// TIA Portal V15.1 export
// export: Created 2024-05-17T05:38:58.0411928Z, ExportSetting WithDefaults, DisplayName Totally Integrated Automation Portal, DisplayVersion V15.1 Update 5, DisplayName TIA Portal Openness, DisplayVersion V15.1 Update 5, DisplayName SINAMICS Startdrive Advanced, DisplayVersion V15.1, DisplayName G130, G150, S120, S150, SINAMICS MV, S210, DisplayVersion V15.1, DisplayName G110M, G120, G120C, G120D, G120P, DisplayVersion V15.1, DisplayName STEP 7 Professional, DisplayVersion V15.1 Update 5, DisplayName STEP 7 Safety, DisplayVersion V15.1, DisplayName WinCC Professional, DisplayVersion V15.1 Update 5, DisplayName SIMATIC Visualization Architect, DisplayVersion V15.1
FUNCTION "209210ZMS012Modes" : Void   // FC311, FBD
TITLE = 209210ZMS012 Modes
{ S7_Optimized_Access := 'FALSE' }
AUTHOR : VCC
FAMILY : Local
NAME : Local
VERSION : 0.1
// stored: AutoNumber false, IsIECCheckEnabled false, SetENOAutomatically False, UDAEnableTagReadback false
   VAR_OUTPUT
      O_AlarmA : Bool;   // Alarm A
      O_AlarmB : Bool;   // Alarm B
      O_AlarmC : Bool;   // Alarm C
      O_AlarmD : Bool;   // Alarm D
      O_AlarmABCondition : Bool;   // Alarms resetable
      H_IAnim : Word;   // Animation bits to Icon in WinCC
   END_VAR
   VAR_TEMP
      NotUsed : Bool;
   END_VAR
BEGIN

REGION Network 1: **** 1 - Inputs **** General Functions
   // General Functions
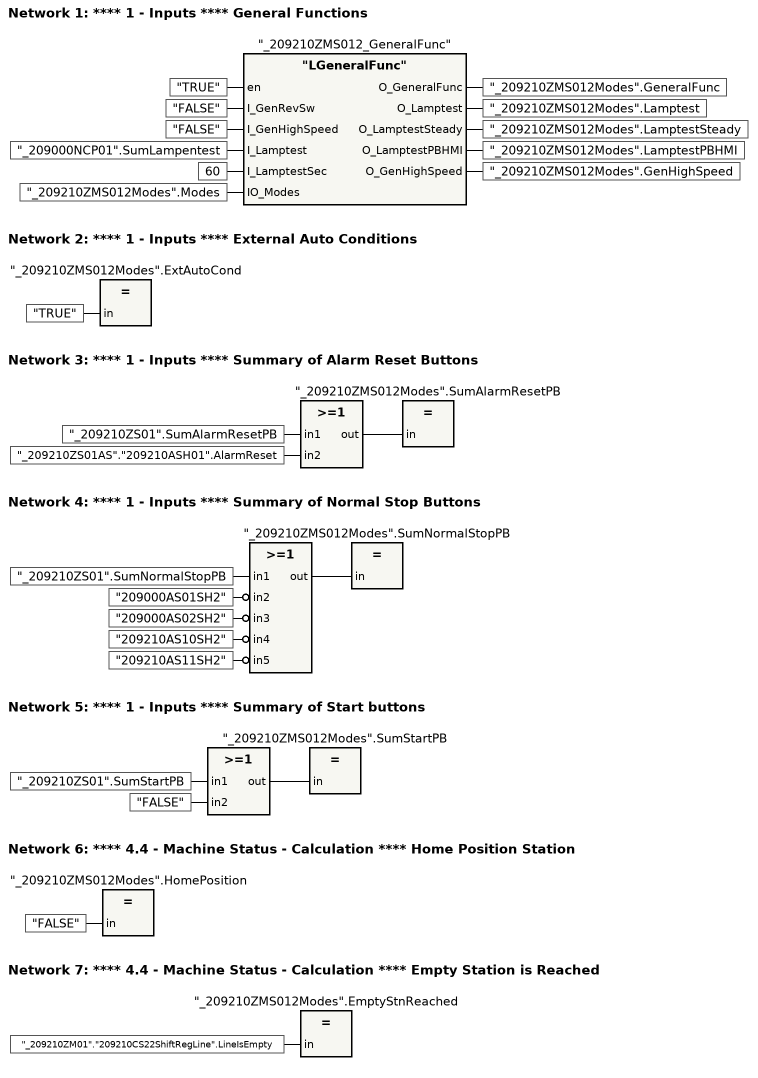
   IF "TRUE" THEN
       "_209210ZMS012_GeneralFunc"(I_GenRevSw := "FALSE",   // "LGeneralFunc"
                               I_GenHighSpeed := "FALSE",
                               I_Lamptest := "_209000NCP01".SumLampentest,
                               I_LamptestSec := 60,
                               IO_Modes := "_209210ZMS012Modes".Modes,
                               O_GeneralFunc => "_209210ZMS012Modes".GeneralFunc,
                               O_Lamptest => "_209210ZMS012Modes".Lamptest,
                               O_LamptestSteady => "_209210ZMS012Modes".LamptestSteady,
                               O_LamptestPBHMI => "_209210ZMS012Modes".LamptestPBHMI,
                               O_GenHighSpeed => "_209210ZMS012Modes".GenHighSpeed);
   END_IF;
END_REGION

REGION Network 2: **** 1 - Inputs **** External Auto Conditions
   "_209210ZMS012Modes".ExtAutoCond := "TRUE";
END_REGION

REGION Network 3: **** 1 - Inputs **** Summary of Alarm Reset Buttons
   // Summary of Alarm Reset Buttons
   "_209210ZMS012Modes".SumAlarmResetPB := "_209210ZS01".SumAlarmResetPB OR "_209210ZS01AS"."209210ASH01".AlarmReset;
END_REGION

REGION Network 4: **** 1 - Inputs **** Summary of Normal Stop Buttons
   // Summary of Normal Stop Buttons
   "_209210ZMS012Modes".SumNormalStopPB := "_209210ZS01".SumNormalStopPB OR NOT "209000AS01SH2" OR NOT "209000AS02SH2" OR NOT "209210AS10SH2" OR NOT "209210AS11SH2";
END_REGION

REGION Network 5: **** 1 - Inputs **** Summary of Start buttons
   // Summary of Start buttons
   "_209210ZMS012Modes".SumStartPB := "_209210ZS01".SumStartPB OR "FALSE";
END_REGION

REGION Network 6: **** 4.4 - Machine Status - Calculation **** Home Position Station
   // Home position
   "_209210ZMS012Modes".HomePosition := "FALSE";
END_REGION

REGION Network 7: **** 4.4 - Machine Status - Calculation **** Empty Station is Reached
   // Empty Station
   "_209210ZMS012Modes".EmptyStnReached := "_209210ZM01"."209210CS22ShiftRegLine".LineIsEmpty;
END_REGION

REGION Network 8: **** 4.5 - Machine Status - Modes **** Mode selector
   // Mode selector
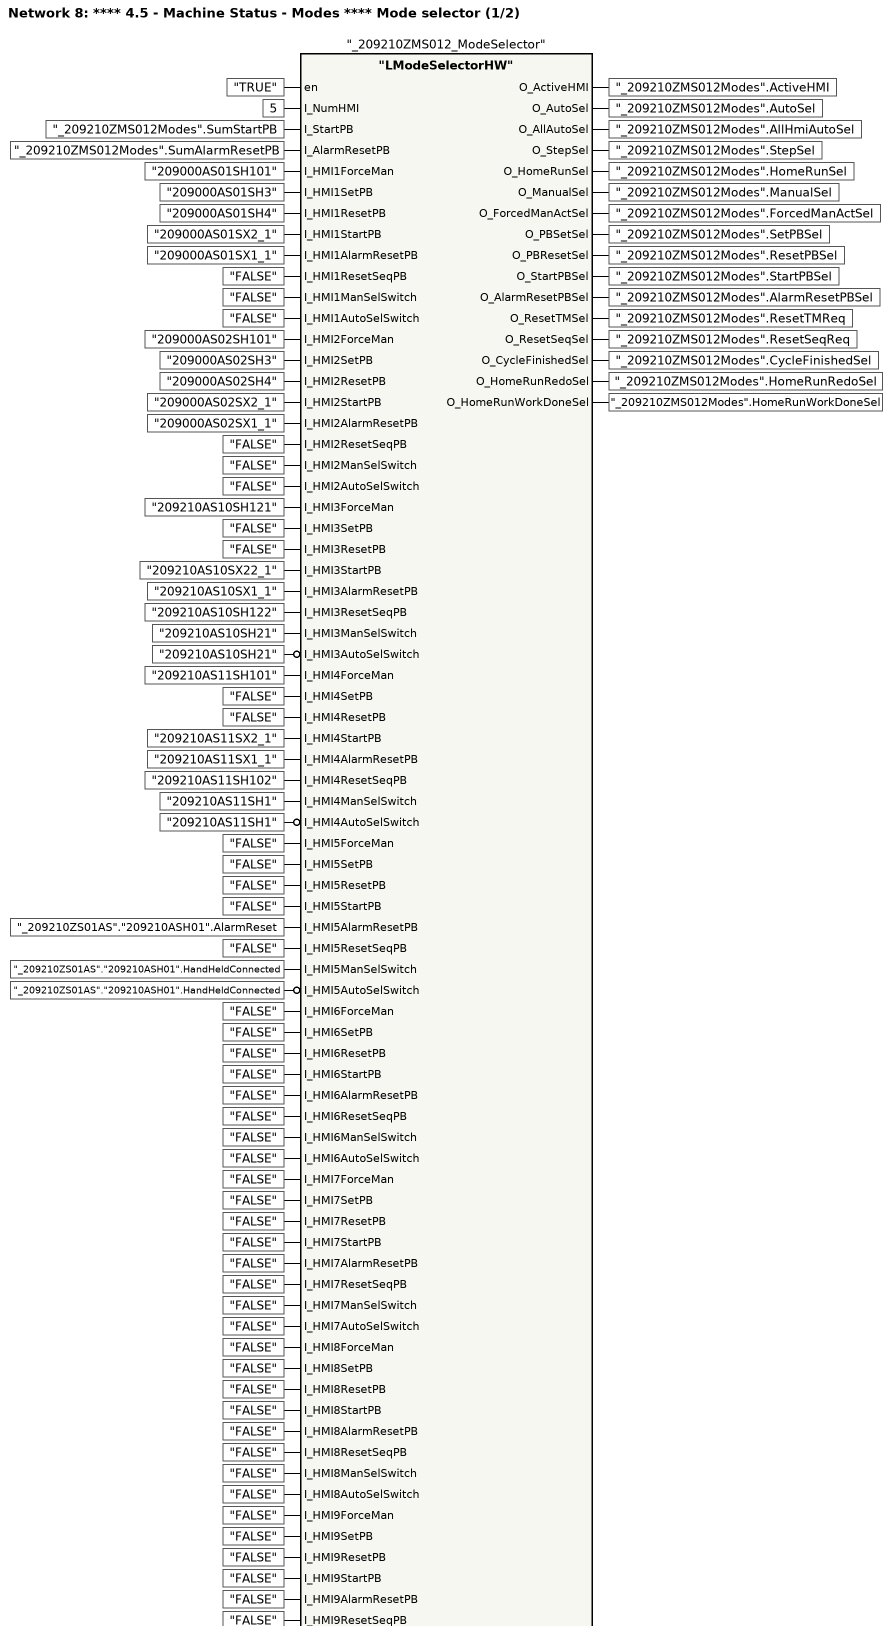
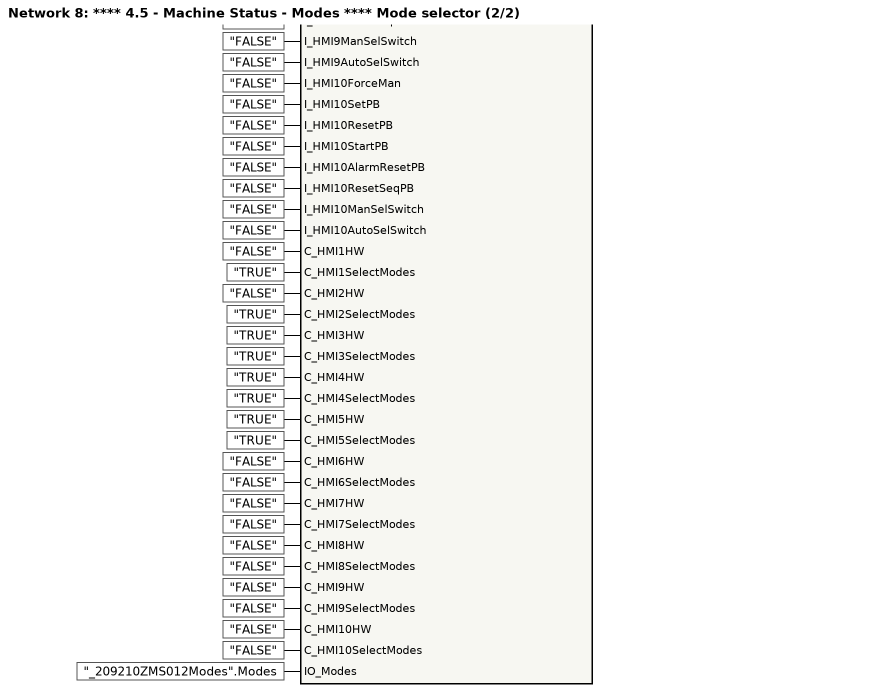
   IF "TRUE" THEN
       "_209210ZMS012_ModeSelector"(I_NumHMI := 5,   // "LModeSelectorHW"
                               I_StartPB := "_209210ZMS012Modes".SumStartPB,
                               I_AlarmResetPB := "_209210ZMS012Modes".SumAlarmResetPB,
                               I_HMI1ForceMan := "209000AS01SH101",
                               I_HMI1SetPB := "209000AS01SH3",
                               I_HMI1ResetPB := "209000AS01SH4",
                               I_HMI1StartPB := "209000AS01SX2_1",
                               I_HMI1AlarmResetPB := "209000AS01SX1_1",
                               I_HMI1ResetSeqPB := "FALSE",
                               I_HMI1ManSelSwitch := "FALSE",
                               I_HMI1AutoSelSwitch := "FALSE",
                               I_HMI2ForceMan := "209000AS02SH101",
                               I_HMI2SetPB := "209000AS02SH3",
                               I_HMI2ResetPB := "209000AS02SH4",
                               I_HMI2StartPB := "209000AS02SX2_1",
                               I_HMI2AlarmResetPB := "209000AS02SX1_1",
                               I_HMI2ResetSeqPB := "FALSE",
                               I_HMI2ManSelSwitch := "FALSE",
                               I_HMI2AutoSelSwitch := "FALSE",
                               I_HMI3ForceMan := "209210AS10SH121",
                               I_HMI3SetPB := "FALSE",
                               I_HMI3ResetPB := "FALSE",
                               I_HMI3StartPB := "209210AS10SX22_1",
                               I_HMI3AlarmResetPB := "209210AS10SX1_1",
                               I_HMI3ResetSeqPB := "209210AS10SH122",
                               I_HMI3ManSelSwitch := "209210AS10SH21",
                               I_HMI3AutoSelSwitch := NOT "209210AS10SH21",
                               I_HMI4ForceMan := "209210AS11SH101",
                               I_HMI4SetPB := "FALSE",
                               I_HMI4ResetPB := "FALSE",
                               I_HMI4StartPB := "209210AS11SX2_1",
                               I_HMI4AlarmResetPB := "209210AS11SX1_1",
                               I_HMI4ResetSeqPB := "209210AS11SH102",
                               I_HMI4ManSelSwitch := "209210AS11SH1",
                               I_HMI4AutoSelSwitch := NOT "209210AS11SH1",
                               I_HMI5ForceMan := "FALSE",
                               I_HMI5SetPB := "FALSE",
                               I_HMI5ResetPB := "FALSE",
                               I_HMI5StartPB := "FALSE",
                               I_HMI5AlarmResetPB := "_209210ZS01AS"."209210ASH01".AlarmReset,
                               I_HMI5ResetSeqPB := "FALSE",
                               I_HMI5ManSelSwitch := "_209210ZS01AS"."209210ASH01".HandHeldConnected,
                               I_HMI5AutoSelSwitch := NOT "_209210ZS01AS"."209210ASH01".HandHeldConnected,
                               I_HMI6ForceMan := "FALSE",
                               I_HMI6SetPB := "FALSE",
                               I_HMI6ResetPB := "FALSE",
                               I_HMI6StartPB := "FALSE",
                               I_HMI6AlarmResetPB := "FALSE",
                               I_HMI6ResetSeqPB := "FALSE",
                               I_HMI6ManSelSwitch := "FALSE",
                               I_HMI6AutoSelSwitch := "FALSE",
                               I_HMI7ForceMan := "FALSE",
                               I_HMI7SetPB := "FALSE",
                               I_HMI7ResetPB := "FALSE",
                               I_HMI7StartPB := "FALSE",
                               I_HMI7AlarmResetPB := "FALSE",
                               I_HMI7ResetSeqPB := "FALSE",
                               I_HMI7ManSelSwitch := "FALSE",
                               I_HMI7AutoSelSwitch := "FALSE",
                               I_HMI8ForceMan := "FALSE",
                               I_HMI8SetPB := "FALSE",
                               I_HMI8ResetPB := "FALSE",
                               I_HMI8StartPB := "FALSE",
                               I_HMI8AlarmResetPB := "FALSE",
                               I_HMI8ResetSeqPB := "FALSE",
                               I_HMI8ManSelSwitch := "FALSE",
                               I_HMI8AutoSelSwitch := "FALSE",
                               I_HMI9ForceMan := "FALSE",
                               I_HMI9SetPB := "FALSE",
                               I_HMI9ResetPB := "FALSE",
                               I_HMI9StartPB := "FALSE",
                               I_HMI9AlarmResetPB := "FALSE",
                               I_HMI9ResetSeqPB := "FALSE",
                               I_HMI9ManSelSwitch := "FALSE",
                               I_HMI9AutoSelSwitch := "FALSE",
                               I_HMI10ForceMan := "FALSE",
                               I_HMI10SetPB := "FALSE",
                               I_HMI10ResetPB := "FALSE",
                               I_HMI10StartPB := "FALSE",
                               I_HMI10AlarmResetPB := "FALSE",
                               I_HMI10ResetSeqPB := "FALSE",
                               I_HMI10ManSelSwitch := "FALSE",
                               I_HMI10AutoSelSwitch := "FALSE",
                               C_HMI1HW := "FALSE",
                               C_HMI1SelectModes := "TRUE",
                               C_HMI2HW := "FALSE",
                               C_HMI2SelectModes := "TRUE",
                               C_HMI3HW := "TRUE",
                               C_HMI3SelectModes := "TRUE",
                               C_HMI4HW := "TRUE",
                               C_HMI4SelectModes := "TRUE",
                               C_HMI5HW := "TRUE",
                               C_HMI5SelectModes := "TRUE",
                               C_HMI6HW := "FALSE",
                               C_HMI6SelectModes := "FALSE",
                               C_HMI7HW := "FALSE",
                               C_HMI7SelectModes := "FALSE",
                               C_HMI8HW := "FALSE",
                               C_HMI8SelectModes := "FALSE",
                               C_HMI9HW := "FALSE",
                               C_HMI9SelectModes := "FALSE",
                               C_HMI10HW := "FALSE",
                               C_HMI10SelectModes := "FALSE",
                               IO_Modes := "_209210ZMS012Modes".Modes,
                               O_ActiveHMI => "_209210ZMS012Modes".ActiveHMI,
                               O_AutoSel => "_209210ZMS012Modes".AutoSel,
                               O_AllAutoSel => "_209210ZMS012Modes".AllHmiAutoSel,
                               O_StepSel => "_209210ZMS012Modes".StepSel,
                               O_HomeRunSel => "_209210ZMS012Modes".HomeRunSel,
                               O_ManualSel => "_209210ZMS012Modes".ManualSel,
                               O_ForcedManActSel => "_209210ZMS012Modes".ForcedManActSel,
                               O_PBSetSel => "_209210ZMS012Modes".SetPBSel,
                               O_PBResetSel => "_209210ZMS012Modes".ResetPBSel,
                               O_StartPBSel => "_209210ZMS012Modes".StartPBSel,
                               O_AlarmResetPBSel => "_209210ZMS012Modes".AlarmResetPBSel,
                               O_ResetTMSel => "_209210ZMS012Modes".ResetTMReq,
                               O_ResetSeqSel => "_209210ZMS012Modes".ResetSeqReq,
                               O_CycleFinishedSel => "_209210ZMS012Modes".CycleFinishedSel,
                               O_HomeRunRedoSel => "_209210ZMS012Modes".HomeRunRedoSel,
                               O_HomeRunWorkDoneSel => "_209210ZMS012Modes".HomeRunWorkDoneSel);
   END_IF;
END_REGION

REGION Network 9: **** 4.5 - Machine Status - Modes **** Modes
   // Modes
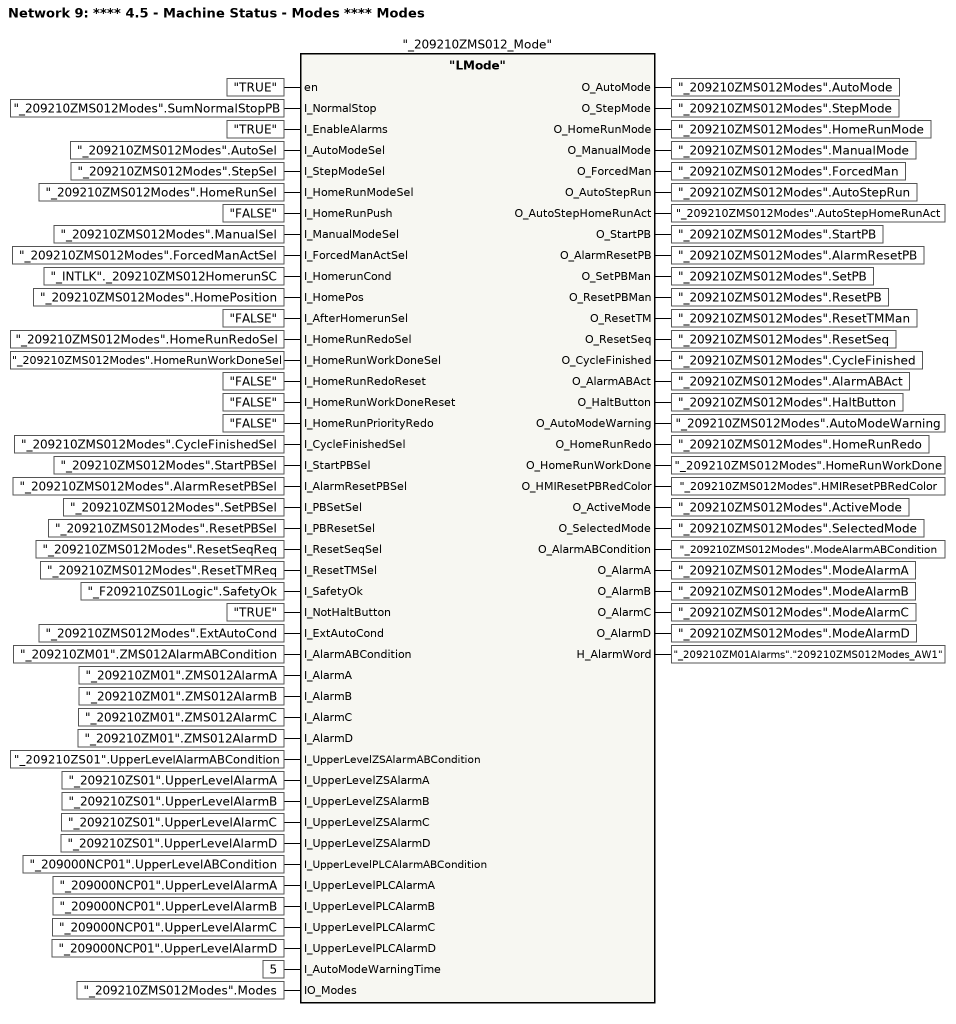
   IF "TRUE" THEN
       "_209210ZMS012_Mode"(I_NormalStop := "_209210ZMS012Modes".SumNormalStopPB,   // "LMode"
                            I_EnableAlarms := "TRUE",
                            I_AutoModeSel := "_209210ZMS012Modes".AutoSel,
                            I_StepModeSel := "_209210ZMS012Modes".StepSel,
                            I_HomeRunModeSel := "_209210ZMS012Modes".HomeRunSel,
                            I_HomeRunPush := "FALSE",
                            I_ManualModeSel := "_209210ZMS012Modes".ManualSel,
                            I_ForcedManActSel := "_209210ZMS012Modes".ForcedManActSel,
                            I_HomerunCond := "_INTLK"._209210ZMS012HomerunSC,
                            I_HomePos := "_209210ZMS012Modes".HomePosition,
                            I_AfterHomerunSel := "FALSE",
                            I_HomeRunRedoSel := "_209210ZMS012Modes".HomeRunRedoSel,
                            I_HomeRunWorkDoneSel := "_209210ZMS012Modes".HomeRunWorkDoneSel,
                            I_HomeRunRedoReset := "FALSE",
                            I_HomeRunWorkDoneReset := "FALSE",
                            I_HomeRunPriorityRedo := "FALSE",
                            I_CycleFinishedSel := "_209210ZMS012Modes".CycleFinishedSel,
                            I_StartPBSel := "_209210ZMS012Modes".StartPBSel,
                            I_AlarmResetPBSel := "_209210ZMS012Modes".AlarmResetPBSel,
                            I_PBSetSel := "_209210ZMS012Modes".SetPBSel,
                            I_PBResetSel := "_209210ZMS012Modes".ResetPBSel,
                            I_ResetSeqSel := "_209210ZMS012Modes".ResetSeqReq,
                            I_ResetTMSel := "_209210ZMS012Modes".ResetTMReq,
                            I_SafetyOk := "_F209210ZS01Logic".SafetyOk,
                            I_NotHaltButton := "TRUE",
                            I_ExtAutoCond := "_209210ZMS012Modes".ExtAutoCond,
                            I_AlarmABCondition := "_209210ZM01".ZMS012AlarmABCondition,
                            I_AlarmA := "_209210ZM01".ZMS012AlarmA,
                            I_AlarmB := "_209210ZM01".ZMS012AlarmB,
                            I_AlarmC := "_209210ZM01".ZMS012AlarmC,
                            I_AlarmD := "_209210ZM01".ZMS012AlarmD,
                            I_UpperLevelZSAlarmABCondition := "_209210ZS01".UpperLevelAlarmABCondition,
                            I_UpperLevelZSAlarmA := "_209210ZS01".UpperLevelAlarmA,
                            I_UpperLevelZSAlarmB := "_209210ZS01".UpperLevelAlarmB,
                            I_UpperLevelZSAlarmC := "_209210ZS01".UpperLevelAlarmC,
                            I_UpperLevelZSAlarmD := "_209210ZS01".UpperLevelAlarmD,
                            I_UpperLevelPLCAlarmABCondition := "_209000NCP01".UpperLevelABCondition,
                            I_UpperLevelPLCAlarmA := "_209000NCP01".UpperLevelAlarmA,
                            I_UpperLevelPLCAlarmB := "_209000NCP01".UpperLevelAlarmB,
                            I_UpperLevelPLCAlarmC := "_209000NCP01".UpperLevelAlarmC,
                            I_UpperLevelPLCAlarmD := "_209000NCP01".UpperLevelAlarmD,
                            I_AutoModeWarningTime := 5,
                            IO_Modes := "_209210ZMS012Modes".Modes,
                            O_AutoMode => "_209210ZMS012Modes".AutoMode,
                            O_StepMode => "_209210ZMS012Modes".StepMode,
                            O_HomeRunMode => "_209210ZMS012Modes".HomeRunMode,
                            O_ManualMode => "_209210ZMS012Modes".ManualMode,
                            O_ForcedMan => "_209210ZMS012Modes".ForcedMan,
                            O_AutoStepRun => "_209210ZMS012Modes".AutoStepRun,
                            O_AutoStepHomeRunAct => "_209210ZMS012Modes".AutoStepHomeRunAct,
                            O_StartPB => "_209210ZMS012Modes".StartPB,
                            O_AlarmResetPB => "_209210ZMS012Modes".AlarmResetPB,
                            O_SetPBMan => "_209210ZMS012Modes".SetPB,
                            O_ResetPBMan => "_209210ZMS012Modes".ResetPB,
                            O_ResetTM => "_209210ZMS012Modes".ResetTMMan,
                            O_ResetSeq => "_209210ZMS012Modes".ResetSeq,
                            O_CycleFinished => "_209210ZMS012Modes".CycleFinished,
                            O_AlarmABAct => "_209210ZMS012Modes".AlarmABAct,
                            O_HaltButton => "_209210ZMS012Modes".HaltButton,
                            O_AutoModeWarning => "_209210ZMS012Modes".AutoModeWarning,
                            O_HomeRunRedo => "_209210ZMS012Modes".HomeRunRedo,
                            O_HomeRunWorkDone => "_209210ZMS012Modes".HomeRunWorkDone,
                            O_HMIResetPBRedColor => "_209210ZMS012Modes".HMIResetPBRedColor,
                            O_ActiveMode => "_209210ZMS012Modes".ActiveMode,
                            O_SelectedMode => "_209210ZMS012Modes".SelectedMode,
                            O_AlarmABCondition => "_209210ZMS012Modes".ModeAlarmABCondition,
                            O_AlarmA => "_209210ZMS012Modes".ModeAlarmA,
                            O_AlarmB => "_209210ZMS012Modes".ModeAlarmB,
                            O_AlarmC => "_209210ZMS012Modes".ModeAlarmC,
                            O_AlarmD => "_209210ZMS012Modes".ModeAlarmD,
                            H_AlarmWord => "_209210ZM01Alarms"."209210ZMS012Modes_AW1");
   END_IF;
END_REGION

REGION Network 10: **** 4.5 - Machine Status - Modes **** Production Modes
   // Production Modes
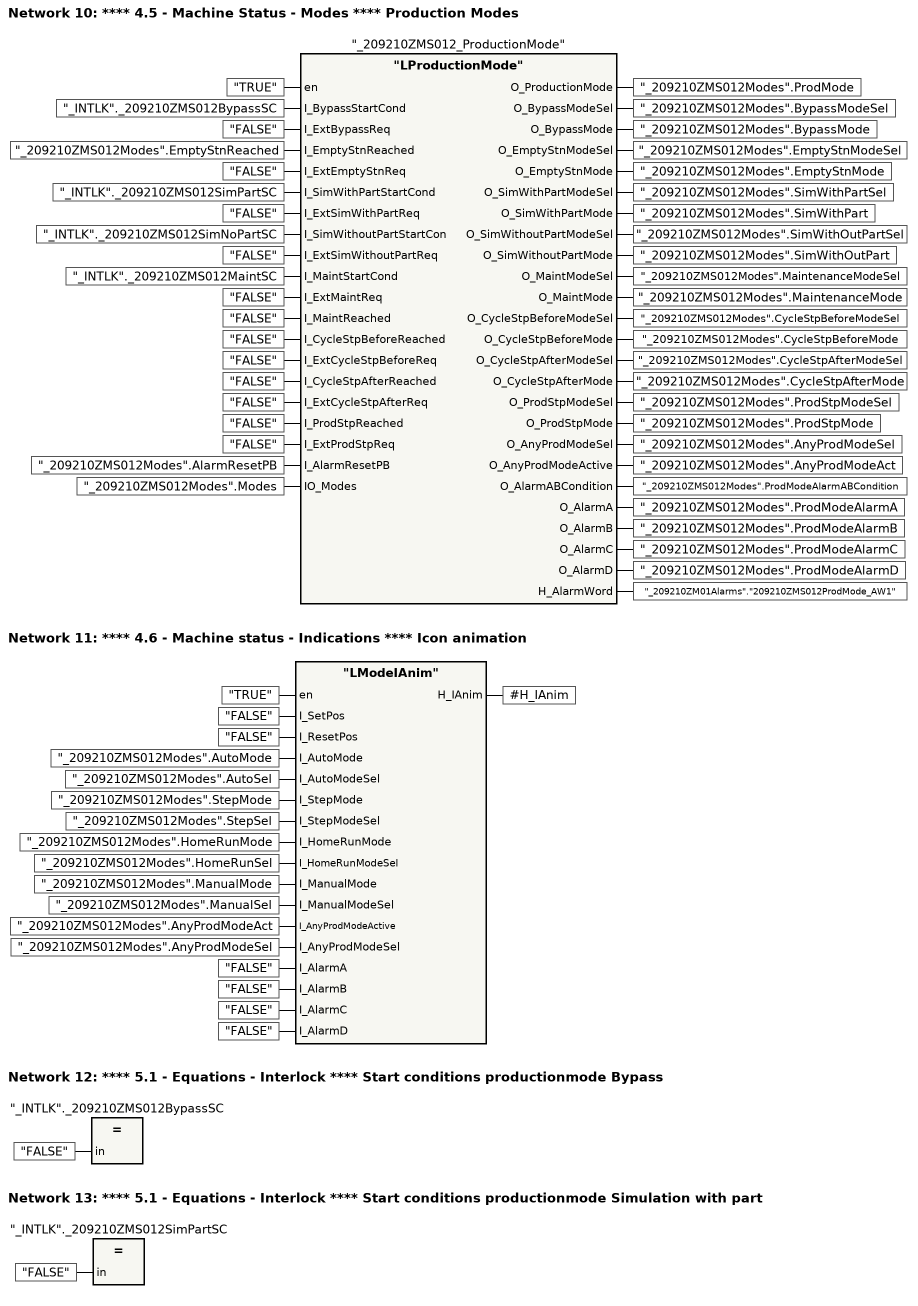
   IF "TRUE" THEN
       "_209210ZMS012_ProductionMode"(I_BypassStartCond := "_INTLK"._209210ZMS012BypassSC,   // "LProductionMode"
                               I_ExtBypassReq := "FALSE",
                               I_EmptyStnReached := "_209210ZMS012Modes".EmptyStnReached,
                               I_ExtEmptyStnReq := "FALSE",
                               I_SimWithPartStartCond := "_INTLK"._209210ZMS012SimPartSC,
                               I_ExtSimWithPartReq := "FALSE",
                               I_SimWithoutPartStartCon := "_INTLK"._209210ZMS012SimNoPartSC,
                               I_ExtSimWithoutPartReq := "FALSE",
                               I_MaintStartCond := "_INTLK"._209210ZMS012MaintSC,
                               I_ExtMaintReq := "FALSE",
                               I_MaintReached := "FALSE",
                               I_CycleStpBeforeReached := "FALSE",
                               I_ExtCycleStpBeforeReq := "FALSE",
                               I_CycleStpAfterReached := "FALSE",
                               I_ExtCycleStpAfterReq := "FALSE",
                               I_ProdStpReached := "FALSE",
                               I_ExtProdStpReq := "FALSE",
                               I_AlarmResetPB := "_209210ZMS012Modes".AlarmResetPB,
                               IO_Modes := "_209210ZMS012Modes".Modes,
                               O_ProductionMode => "_209210ZMS012Modes".ProdMode,
                               O_BypassModeSel => "_209210ZMS012Modes".BypassModeSel,
                               O_BypassMode => "_209210ZMS012Modes".BypassMode,
                               O_EmptyStnModeSel => "_209210ZMS012Modes".EmptyStnModeSel,
                               O_EmptyStnMode => "_209210ZMS012Modes".EmptyStnMode,
                               O_SimWithPartModeSel => "_209210ZMS012Modes".SimWithPartSel,
                               O_SimWithPartMode => "_209210ZMS012Modes".SimWithPart,
                               O_SimWithoutPartModeSel => "_209210ZMS012Modes".SimWithOutPartSel,
                               O_SimWithoutPartMode => "_209210ZMS012Modes".SimWithOutPart,
                               O_MaintModeSel => "_209210ZMS012Modes".MaintenanceModeSel,
                               O_MaintMode => "_209210ZMS012Modes".MaintenanceMode,
                               O_CycleStpBeforeModeSel => "_209210ZMS012Modes".CycleStpBeforeModeSel,
                               O_CycleStpBeforeMode => "_209210ZMS012Modes".CycleStpBeforeMode,
                               O_CycleStpAfterModeSel => "_209210ZMS012Modes".CycleStpAfterModeSel,
                               O_CycleStpAfterMode => "_209210ZMS012Modes".CycleStpAfterMode,
                               O_ProdStpModeSel => "_209210ZMS012Modes".ProdStpModeSel,
                               O_ProdStpMode => "_209210ZMS012Modes".ProdStpMode,
                               O_AnyProdModeSel => "_209210ZMS012Modes".AnyProdModeSel,
                               O_AnyProdModeActive => "_209210ZMS012Modes".AnyProdModeAct,
                               O_AlarmABCondition => "_209210ZMS012Modes".ProdModeAlarmABCondition,
                               O_AlarmA => "_209210ZMS012Modes".ProdModeAlarmA,
                               O_AlarmB => "_209210ZMS012Modes".ProdModeAlarmB,
                               O_AlarmC => "_209210ZMS012Modes".ProdModeAlarmC,
                               O_AlarmD => "_209210ZMS012Modes".ProdModeAlarmD,
                               H_AlarmWord => "_209210ZM01Alarms"."209210ZMS012ProdMode_AW1");
   END_IF;
END_REGION

REGION Network 11: **** 4.6 - Machine status - Indications **** Icon animation
   // Icon animation
   IF "TRUE" THEN
       "LModeIAnim"(I_SetPos := "FALSE",
                    I_ResetPos := "FALSE",
                    I_AutoMode := "_209210ZMS012Modes".AutoMode,
                    I_AutoModeSel := "_209210ZMS012Modes".AutoSel,
                    I_StepMode := "_209210ZMS012Modes".StepMode,
                    I_StepModeSel := "_209210ZMS012Modes".StepSel,
                    I_HomeRunMode := "_209210ZMS012Modes".HomeRunMode,
                    I_HomeRunModeSel := "_209210ZMS012Modes".HomeRunSel,
                    I_ManualMode := "_209210ZMS012Modes".ManualMode,
                    I_ManualModeSel := "_209210ZMS012Modes".ManualSel,
                    I_AnyProdModeActive := "_209210ZMS012Modes".AnyProdModeAct,
                    I_AnyProdModeSel := "_209210ZMS012Modes".AnyProdModeSel,
                    I_AlarmA := "FALSE",
                    I_AlarmB := "FALSE",
                    I_AlarmC := "FALSE",
                    I_AlarmD := "FALSE",
                    H_IAnim => #H_IAnim);
   END_IF;
END_REGION

REGION Network 12: **** 5.1 - Equations - Interlock **** Start conditions productionmode Bypass
   // Start conditions productionmode
   // Bypass
   "_INTLK"._209210ZMS012BypassSC := "FALSE";
END_REGION

REGION Network 13: **** 5.1 - Equations - Interlock **** Start conditions productionmode Simulation with part
   // Start conditions productionmode
   // Simulation with part
   "_INTLK"._209210ZMS012SimPartSC := "FALSE";
END_REGION

REGION Network 14: **** 5.1 - Equations - Interlock **** Start conditions productionmode Simulation without part
   // Start conditions productionmode
   // Simulation without part
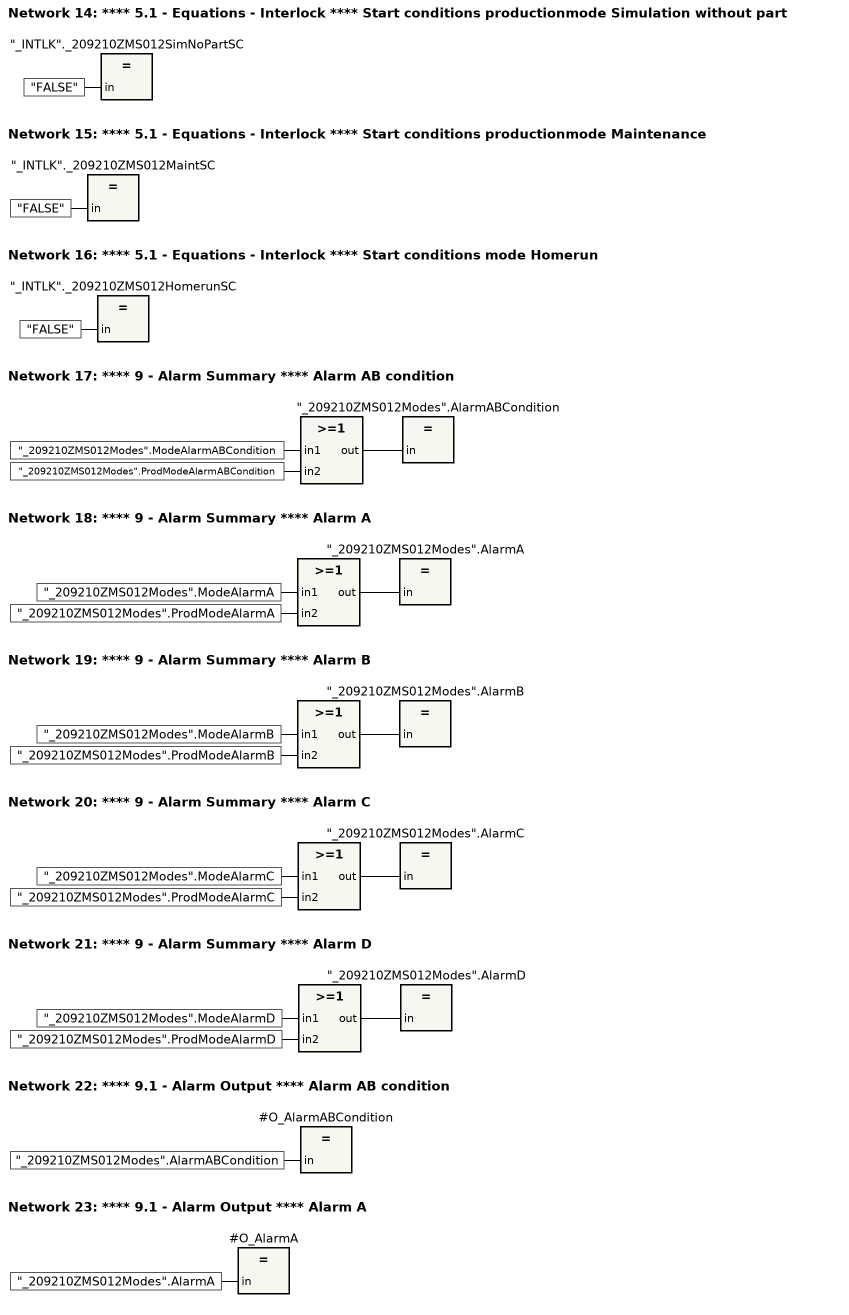
   "_INTLK"._209210ZMS012SimNoPartSC := "FALSE";
END_REGION

REGION Network 15: **** 5.1 - Equations - Interlock **** Start conditions productionmode Maintenance
   // Start conditions productionmode
   // Maintenance
   "_INTLK"._209210ZMS012MaintSC := "FALSE";
END_REGION

REGION Network 16: **** 5.1 - Equations - Interlock **** Start conditions mode Homerun
   // Start conditions mode
   // Homerun
   "_INTLK"._209210ZMS012HomerunSC := "FALSE";
END_REGION

REGION Network 17: **** 9 - Alarm Summary **** Alarm AB condition
   // Alarm AB condition
   "_209210ZMS012Modes".AlarmABCondition := "_209210ZMS012Modes".ModeAlarmABCondition OR "_209210ZMS012Modes".ProdModeAlarmABCondition;
END_REGION

REGION Network 18: **** 9 - Alarm Summary **** Alarm A
   // Summary of alarms A
   "_209210ZMS012Modes".AlarmA := "_209210ZMS012Modes".ModeAlarmA OR "_209210ZMS012Modes".ProdModeAlarmA;
END_REGION

REGION Network 19: **** 9 - Alarm Summary **** Alarm B
   // Summary of alarms B
   "_209210ZMS012Modes".AlarmB := "_209210ZMS012Modes".ModeAlarmB OR "_209210ZMS012Modes".ProdModeAlarmB;
END_REGION

REGION Network 20: **** 9 - Alarm Summary **** Alarm C
   // Summary of alarms C
   "_209210ZMS012Modes".AlarmC := "_209210ZMS012Modes".ModeAlarmC OR "_209210ZMS012Modes".ProdModeAlarmC;
END_REGION

REGION Network 21: **** 9 - Alarm Summary **** Alarm D
   // Summary of alarms D
   "_209210ZMS012Modes".AlarmD := "_209210ZMS012Modes".ModeAlarmD OR "_209210ZMS012Modes".ProdModeAlarmD;
END_REGION

REGION Network 22: **** 9.1 - Alarm Output **** Alarm AB condition
   // Alarm AB condition
   #O_AlarmABCondition := "_209210ZMS012Modes".AlarmABCondition;
END_REGION

REGION Network 23: **** 9.1 - Alarm Output **** Alarm A
   // Summary of alarms A
   #O_AlarmA := "_209210ZMS012Modes".AlarmA;
END_REGION

REGION Network 24: **** 9.1 - Alarm Output **** Alarm B
   // Summary of alarms B
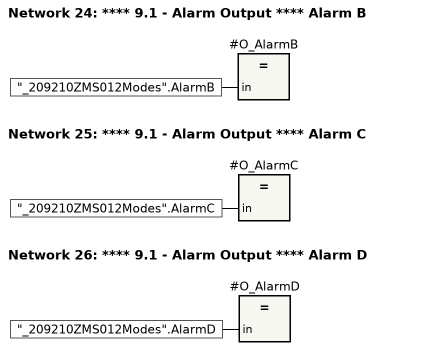
   #O_AlarmB := "_209210ZMS012Modes".AlarmB;
END_REGION

REGION Network 25: **** 9.1 - Alarm Output **** Alarm C
   // Summary of alarms C
   #O_AlarmC := "_209210ZMS012Modes".AlarmC;
END_REGION

REGION Network 26: **** 9.1 - Alarm Output **** Alarm D
   // Summary of alarms D
   #O_AlarmD := "_209210ZMS012Modes".AlarmD;
END_REGION
END_FUNCTION
